// TIA Portal V17 export
// export: Created 2023-02-14T02:49:50.3483306Z, ExportSetting WithDefaults, DisplayName Totally Integrated Automation Portal, DisplayVersion V17, DisplayName TIA Portal Openness, DisplayVersion V17, DisplayName TIA Portal Teamcenter Gateway, DisplayVersion V17, DisplayName TIA Portal Version Control Interface, DisplayVersion V17, DisplayName SINAMICS Startdrive Advanced, DisplayVersion V17, DisplayName SINAMICS Startdrive G130, G150, S120, S150, SINAMICS MV, S210, DisplayVersion V17, DisplayName SINAMICS Startdrive G110M, G120, G120C, G120D, G120P, G115D, DisplayVersion V17, DisplayName STEP 7 Professional, DisplayVersion V17, DisplayName STEP 7 Safety, DisplayVersion V17, DisplayName WinCC Professional, DisplayVersion V17
DATA_BLOCK "T-04.01_DB"   // DB354
VERSION : 0.1
// stored: AutoNumber false, DBAccessibleFromOPCUA true, DBAccessibleFromWebserver true, InstanceOfName BFT_Type1, InstanceOfType FB
"BFT_Type1"
   // VAR_INPUT
   //    "IN_FBAV.01" : Bool;
   //    "IN_FBAV.02" : Bool;
   //    "IN_FBAV.03" : Bool;
   //    "IN_FBAV.04" : Bool;
   //    "IN_FBAV.05" : Bool;
   //    "IN_FBAV.06" : Bool;
   //    "IN_FBAV.07" : Bool;
   //    "IN_FBAV.08" : Bool;
   //    "IN_FBAV.09" : Bool;
   //    IN_LT01 : Real;
   //    "IN_FBP.01" : Bool;
   //    "IN_P.01-Speed" : Real;
   //    "IN_FBP.02" : Bool;
   //    "IN_P.02-Speed" : Real;
   //    "IN_FBP.03" : Bool;
   //    "IN_P.03-Speed" : Real;
   //    DosePumpSpeed : Real;
   //    "DoseON-OFF" : Bool;
   //    "DosePumpON-OFF" : Bool;
   //    CIPPulse : Bool;
   //    CIP_Supply_ON : Bool;
   //    LineTrf_OK : Bool;
   //    LineFlush_OK : Bool;
   //    Loading_Busy : Bool;
   // END_VAR
   // VAR_OUTPUT
   //    "OUT_AV.01" : Bool;
   //    "OUT_AV.02" : Bool;
   //    "OUT_AV.03" : Bool;
   //    "OUT_AV.04" : Bool;
   //    "OUT_AV.05" : Bool;
   //    "OUT_AV.06" : Bool;
   //    "OUT_AV.07" : Bool;
   //    "OUT_AV.08" : Bool;
   //    "OUT_AV.09" : Bool;
   //    "OUT_P.01" : Bool;
   //    "OUT_P.01-Speed" : Real;
   //    "OUT_P.02" : Bool;
   //    "OUT_P.02-Speed" : Real;
   //    "OUT_P.03" : Bool;
   //    "OUT_P.03-Speed" : Real;
   //    OUT_CIPTank_AVOpen : Bool;
   //    OUT_CIPLine_AVOpen : Bool;
   // END_VAR
   // VAR
   //    Cmd : Struct
   //       Inload : Bool;
   //       Tank_CIP_Req : Bool;
   //       Line_CIP_Req : Bool;
   //       Flushing : Bool;
   //       RaadyForMix : Bool;
   //       Flush_Select : Byte;
   //    END_STRUCT;
   //    Param : Struct
   //       SP_Level_LL : Real;
   //       SP_Level_ML : Real;
   //       SP_Level_HL : Real;
   //       SupplyPump_SP_Speed : Real;
   //       L_Hi_Lim : Real;
   //       L_Lo_Lim : Real;
   //       L_Hys : Real;
   //       FlushingTime : DInt;
   //       CIP_Trf_SP_Speed : Real;
   //       CIP_Ret_ON_SP : Real;
   //       CIP_Ret_OFF_SP : Real;
   //    END_STRUCT;
   //    State : Struct
   //       Tank_inloading : Bool;
   //       Tank_inCIP : Bool;
   //       Line_inCIP : Bool;
   //       Flushing : Bool;
   //       Tank_LL : Bool;
   //       Tank_ML : Bool;
   //       Tank_HL : Bool;
   //       Inload_Enable : Bool;
   //       Tank_CIP_Enable : Bool;
   //       Line_CIP_Enable : Bool;
   //       Flushing_Enable : Bool;
   //       Flush_selected : Byte;
   //       CIP_Request_OK : Bool;
   //       CIP_ReturnON : Bool;
   //       Ready_For_Transfer_EN : Bool;
   //       Ready_For_Transfer : Bool;
   //       HWT_Status : Int;
   //       Transfer_to_Blend : Bool;
   //    END_STRUCT;
   //    alwaysON : Bool;
   //    L_Hys_Abs : Real;
   //    Hys_Level_HL : Real;
   //    Hys_Level_ML : Real;
   //    Hys_Level_LL : Real;
   //    r : Struct
   //       PosE1 : Bool;
   //       PosE2 : Bool;
   //       PosE3 : Bool;
   //       PosE4 : Bool;
   //       PosE5 : Bool;
   //       PosE6 : Bool;
   //       PosE7 : Bool;
   //       PosE8 : Bool;
   //       PosE9 : Bool;
   //       PosE10 : Bool;
   //       PosE11 : Bool;
   //       PosE12 : Bool;
   //       PosE13 : Bool;
   //       PosE14 : Bool;
   //       PosE15 : Bool;
   //       PosE16 : Bool;
   //       PosE17 : Bool;
   //       PosE18 : Bool;
   //       PosE19 : Bool;
   //       PosE20 : Bool;
   //       PosE21 : Bool;
   //       PosE22 : Bool;
   //       PosE23 : Bool;
   //       PosE24 : Bool;
   //       PosE25 : Bool;
   //       PosE26 : Bool;
   //       PosE27 : Bool;
   //       PosE28 : Bool;
   //       PosE29 : Bool;
   //       PosE30 : Bool;
   //       PosE31 : Bool;
   //       PosE32 : Bool;
   //    END_STRUCT;
   //    Actuator : Struct
   //       AV_Outlet : Bool;
   //       TransferPump : Bool;
   //       FlushPump : Bool;
   //       CV_Steam : Bool;
   //       Pump : Bool;
   //    END_STRUCT;
   //    FlushingTim : TON_TIME;
   //    SPumpTim { S7_SetPoint := 'True'} : TON_TIME;
   //    AVinloadTim { S7_SetPoint := 'True'} : TON_TIME;
   // END_VAR
BEGIN
END_DATA_BLOCK
